FUNCTION_BLOCK FB_MotionDrive_Test EXTENDS FB_TestSuite
VAR
    fbMoveRequest : FB_MoveRequest_TestDouble;
    fbEpicsMotionParamsStatus : FB_EpicsMotionParamsStatus_TestDouble;
    fbMotionAxis: FB_MotionAxisNC_TestDouble;
    fbBrake 				: FB_Brake_TestDouble;
    fbMotionInterlocks	: FB_MotionInterlocksLimSw_TestDouble;
    fbMotionLogger 		: FB_MotionLogger_TestDouble;
    fbMotionDriveStateMachine : FB_MotionDriveStateMachine_TestDouble;
END_VAR

NoCrashTest();

METHOD NoCrashTest
VAR_INST
    fbMotionDrive : FB_MotionDrive(
                                    iMotionAxis := fbMotionAxis,
                                    iMotionLogger:=fbMotionLogger,
                                    iBrake:=fbBrake,
                                    iMotionInterlocks:=fbMotionInterlocks,
                                    iMoveRequest :=fbMoveRequest,
                                    iEpicsMotionParamsStatus := fbEpicsMotionParamsStatus,
                                    iMotionDriveStateMachine := fbMotionDriveStateMachine
                                );


END_VAR
(*This method is called cyclicly in the fbMotionDrive *)
TEST(__POUNAME());
fbMotionDrive();
TEST_FINISHED();
END_METHOD

END_FUNCTION_BLOCK

(* stored: Version 1.1.0.1
   POU FB_MotionDrive_Test: Id {fa0c0ca3-2ef2-4761-b316-41cf1af95b88}, SpecialFunc None
   Method NoCrashTest: Id {75361fae-01d6-457b-bd6b-fe3e29169e9e} *)
